FUNCTION_BLOCK Manager IMPLEMENTS I_RegisterMover, I_RegisterPosition
VAR CONSTANT
	MAX_MOVERS 		: INT := 10;
	MAX_POSITIONS	: INT := 10;
END_VAR
VAR
	_IMover 		: ARRAY [1..SETTINGS.MAX_MOVERS] OF I_Mover;
	_moverCount 	: INT;
	_IPos			: ARRAY [1..SETTINGS.MAX_POSITIONS] OF I_Position;
	_PosCount 		: INT;
END_VAR

METHOD PRIVATE _FindUnlinkedMoverWithStep : I_Mover
VAR_INPUT
	MoverStep : UDINT;
END_VAR
VAR
	i : INT;
	IMover : I_Mover;
END_VAR
FOR i:=1 TO _moverCount DO
	IMover := _IMover[i];
	IF IMover <> 0 THEN
		IF IMover.Step = MoverStep AND NOT IMover.Linked THEN
			_FindUnlinkedMoverWithStep := IMover;
		EXIT;	
		END_IF		
	END_IF
END_FOR
END_METHOD

METHOD Cyclic : BOOL
VAR_INPUT
END_VAR
VAR
	i : INT;
	StepRequest : UDINT;
	IMover		: I_Mover;
	IMoverPos 	: I_MoverPos;
	IPos		: I_Position;
END_VAR
// Call Positions
IMover := 0;
FOR i:=1 TO _PosCount DO
	IPos := _IPos[i];
	IF IPos <> 0 THEN
		IF IPos.RequestMover THEN
			IMover := _FindUnlinkedMoverWithStep(Ipos.RequestedStep);
			IF IMover <> 0 THEN
				Ipos.SetMoverLink(IMover);
				IMover.SetPosLink(IPos);	
			END_IF	
		END_IF
	END_IF
END_FOR

// Call Movers
FOR i:=1 TO _moverCount DO
	_IMover[i].Cyclic();
END_FOR
END_METHOD

METHOD RegisterMover : BOOL
VAR_INPUT
	mover : I_Mover;
END_VAR
VAR
	i : INT;
END_VAR
IF _moverCount < SETTINGS.MAX_MOVERS THEN
//	IF mover <> 0 THEN
		_moverCount := _moverCount + 1;
		_IMover[_moverCount] := mover;
		RegisterMover := TRUE;	
//	END_IF
END_IF
END_METHOD

METHOD RegisterPosition : BOOL
VAR_INPUT
	position : I_Position;
END_VAR
VAR
	i : INT;
END_VAR
IF _PosCount < SETTINGS.MAX_POSITIONS THEN
	IF position <> 0 THEN
		_PosCount := _PosCount + 1;
		_IPos[_PosCount] := position;
		RegisterPosition := TRUE;	
	END_IF
END_IF
END_METHOD

END_FUNCTION_BLOCK

(* stored: Version 1.1.0.1
   POU Manager: Id {13c3e8db-89c0-4855-ae61-1add72aaab8d}, SpecialFunc None
   Method _FindUnlinkedMoverWithStep: Id {97ccd672-585d-4765-9d33-7f901e86f746}
   Method Cyclic: Id {2fa8a194-e773-4fee-80d2-3115ff523d3f}
   Method RegisterMover: Id {3f37e71d-6e2f-4dd5-a4e3-6327ddbedb63}
   Method RegisterPosition: Id {9cebef58-b78c-40ca-ab33-33f63a042f35} *)
